Yaskawa INFORM job: R2_W02,4,6(0_0)_MP_OK.JBI

/JOB
//NAME R2_W02,4,6(0_0)_MP_OK
///FOLDERNAME MP_TEST
//POS
///NPOS 87,87,0,4,0,0
///TOOL 0
///POSTYPE PULSE
///PULSE
C00000=174522,6583,732,81114,57384,11781
C00001=174517,6598,745,81115,57387,11780
C00002=174515,6604,750,81115,57388,11780
C00003=173653,9147,2977,81262,57995,11683
C00004=173711,9248,3067,81257,57952,11686
C00005=173653,9147,2977,81262,57995,11683
C00006=174515,6604,750,81115,57388,11780
C00007=174498,6652,791,75592,65380,14408
C00008=174498,6652,791,75592,65380,14408
C00009=174498,6652,791,75592,65380,14408
C00010=176658,117,-15048,82463,49173,12368
C00011=174531,6571,721,88243,49982,8451
C00012=174533,6604,911,88329,49975,8393
C00013=174531,6571,721,88243,49982,8451
C00014=174523,6586,734,88244,49988,8450
C00015=174526,6579,728,88244,49987,8450
C00016=174531,6564,715,88243,49983,8451
C00017=160984,-11348,3930,36053,37207,-42708
C00018=160980,-11334,3941,36055,37209,-42709
C00019=160979,-11329,3945,36056,37210,-42710
C00020=161194,-11069,4145,35902,37129,-42610
C00021=160979,-11329,3945,36056,37210,-42710
C00022=160995,-11368,3914,36742,28122,-41255
C00023=160996,-11216,4319,36932,27985,-41352
C00024=160995,-11368,3914,36742,28122,-41255
C00025=160973,-11311,3958,34758,46261,-43992
C00026=160980,-11331,3943,34756,46258,-43990
C00027=160980,-11331,3943,34756,46258,-43990
C00028=160980,-11331,3943,34756,46258,-43990
C00029=160973,-11311,3958,34758,46261,-43992
C00030=160973,-11311,3958,34758,46261,-43992
C00031=160974,-11316,3955,34758,46261,-43992
C00032=160977,-11328,3945,34757,46259,-43991
C00033=155155,-6207,-30499,23040,84085,-41474
C00034=187974,16007,-465,74860,68606,73739
C00035=187971,16014,-459,74861,68608,73738
C00036=187970,16017,-457,74861,68609,73738
C00037=188065,16322,-175,74847,68538,73741
C00038=187970,16017,-457,74861,68609,73738
C00039=187982,15993,-478,74858,68601,73740
C00040=188123,15688,-759,74825,68507,73762
C00041=187982,15993,-478,74858,68601,73740
C00042=187982,15995,-476,74858,68601,73740
C00043=188055,16230,-74,74890,68512,73687
C00044=187982,15995,-476,74858,68601,73740
C00045=187983,15992,-479,74858,68601,73740
C00046=187985,15986,-485,74857,68599,73740
C00047=155155,-6207,-30499,23040,84085,-41474
C00048=161010,6792,897,39431,61770,-2600
C00049=161008,6803,906,39432,61771,-2600
C00050=161106,6439,785,39434,61637,-2607
C00051=161075,4879,-316,39487,61556,-2657
C00052=160508,6816,-113,39396,62494,-2543
C00053=161011,6899,1448,34591,61140,-1667
C00054=173294,-15772,-2365,19599,41502,-27150
C00055=174899,-11478,4010,19118,39501,-26768
C00056=174262,-12641,3696,19743,39267,-27176
C00057=174084,-11684,2460,19373,40493,-26971
C00058=174842,-11820,3581,23453,38073,-33209
C00059=174431,-11387,3914,23749,38204,-33407
C00060=174436,-11399,3906,23747,38202,-33405
C00061=174416,-11363,3933,23761,38209,-33414
C00062=155155,-6207,-30499,23040,84085,-41474
C00063=174170,40084,30970,44829,89709,-71753
C00064=174201,39824,30698,44830,89717,-71735
C00065=174202,39772,30629,44830,89729,-71730
C00066=174202,39771,30687,44829,89703,-71742
C00067=173753,38726,28593,44851,90472,-71609
C00068=173790,41778,32604,44829,89804,-71890
C00069=174284,39520,30698,43457,86472,-69264
C00070=174527,39515,30359,43444,86501,-69136
C00071=174215,39612,30410,43455,86673,-69209
C00072=174214,39663,30476,43455,86662,-69214
C00073=174184,39924,30747,43457,86653,-69232
C00074=155155,-6207,-30499,23040,84085,-41474
C00075=160633,-10270,5638,28338,22900,-47145
C00076=162219,-15798,1425,26285,22163,-46063
C00077=160659,-10505,5478,28325,22871,-47138
C00078=160661,-10727,4919,28067,23075,-47011
C00079=161098,-12444,3311,27327,23025,-46629
C00080=159658,-10599,5699,29947,23053,-47982
C00081=160917,-11163,4021,24405,19147,-46607
C00082=160969,-11372,4753,24990,18622,-46880
C00083=160661,-10807,5180,25528,18740,-47150
C00084=160656,-10808,5155,25519,18754,-47146
C00085=135615,-20366,-13260,37178,48093,-50762
C00086=15978,-102434,-83816,28834,48298,-44128
BC00000=388510,12234,707895
BC00001=380989,10464,701589
BC00002=377980,9756,699066
BC00003=377846,15,698926
BC00004=375507,15,698920
BC00005=377846,15,698926
BC00006=377980,9756,699066
BC00007=360773,4968,724258
BC00008=360752,2897,724236
BC00009=360773,4968,724258
BC00010=374300,26988,580273
BC00011=374300,26988,580273
BC00012=374302,26995,572208
BC00013=374300,26988,580273
BC00014=379137,9576,654055
BC00015=382103,10646,655203
BC00016=389520,13320,658072
BC00017=313352,46812,968569
BC00018=306234,44848,958660
BC00019=303387,44062,954697
BC00020=300998,44084,954691
BC00021=303387,44062,954697
BC00022=302385,72266,846935
BC00023=302386,72273,838870
BC00024=302385,72266,846935
BC00025=301794,28524,989445
BC00026=305297,28517,959783
BC00027=305280,26764,959765
BC00028=305297,28517,959783
BC00029=301794,28524,989445
BC00030=301708,28983,989449
BC00031=304507,29324,994442
BC00032=311505,30175,1006925
BC00033=296594,86442,873629
BC00034=388565,51804,658383
BC00035=383620,57007,647781
BC00036=381641,59088,643541
BC00037=379252,59110,643535
BC00038=381641,59088,643541
BC00039=390370,60897,618560
BC00040=390394,63201,618584
BC00041=390370,60897,618560
BC00042=388386,59719,612189
BC00043=388387,59726,604124
BC00044=388386,59719,612189
BC00045=390364,57638,616429
BC00046=395310,52435,627031
BC00047=296594,86442,873629
BC00048=313394,73469,855255
BC00049=307271,69988,843128
BC00050=304895,68636,838421
BC00051=304822,68595,838277
BC00052=304822,68595,838277
BC00053=308544,65120,825419
BC00054=314454,36752,936853
BC00055=314454,36752,936853
BC00056=314454,36752,936853
BC00057=314454,36752,936853
BC00058=323351,25201,911905
BC00059=326138,25881,916533
BC00060=333107,27583,928104
BC00061=333060,27580,1035638
BC00062=296594,86442,873629
BC00063=333324,97353,980736
BC00064=333273,97166,873204
BC00065=330544,102864,857707
BC00066=329453,105143,851509
BC00067=329453,105143,851509
BC00068=329453,105143,851509
BC00069=333744,110491,853540
BC00070=351310,110324,799899
BC00071=352593,108156,806169
BC00072=355802,102738,821843
BC00073=355852,102924,929375
BC00074=296594,86442,873629
BC00075=301704,63726,1065666
BC00076=301654,63540,958133
BC00077=294938,60391,948793
BC00078=292251,59131,945057
BC00079=292251,59131,945057
BC00080=292251,59131,945057
BC00081=289814,66040,921083
BC00082=289884,78172,833466
BC00083=292523,79582,836925
BC00084=299118,83106,845574
BC00085=299169,83292,953107
BC00086=277147,104204,968203
///POSTYPE BASE
///RECTAN
///RCONF 0,0,0,0,0,0,0,0,0,0,0,0,0,0,0,0,0,0,0,0,0,0,0,0
P00006=0.222,-3.123,-1.508,0.0000,0.0000,0.0000
P00021=-0.225,-6.128,-0.405,0.0000,0.0000,0.0000
P00024=0.145,-0.552,1.326,0.0000,0.0000,0.0000
P00026=0.562,-0.002,-0.337,0.0000,0.0000,0.0000
//INST
///DATE 2023/11/16 16:40
///ATTR SC,RW
///GROUP1 RB1,BS1
NOP
'r2_W02,4,6
'Path S702 (for W1)
SFTOF
MOVL C00000 BC00000 V=100.0
MOVL C00001 BC00001 V=100.0
MOVL C00002 BC00002 V=100.0
MOVL C00003 BC00003 V=60.0
REFP 3 C00004 BC00004
CALL JOB:SEARCH-R1
SET P021 P006
SFTON P021
MOVL C00005 BC00005 V=60.0
MOVL C00006 BC00006 V=100.0
MOVL C00007 BC00007 V=60.0
REFP 3 C00008 BC00008
CALL JOB:SEARCH-R1
SET P021 P006
SFTON P021
MOVL C00009 BC00009 V=60.0
MOVL C00010 BC00010 V=100.0
MOVL C00011 BC00011 V=60.0
REFP 3 C00012 BC00012
CALL JOB:SEARCH-R1
SET P021 P006
SFTON P021
MOVL C00013 BC00013 V=60.0
MOVL C00014 BC00014 V=100.0
MOVL C00015 BC00015 V=100.0
MOVL C00016 BC00016 V=100.0
'Path S708 (for W4)
SFTOF
MOVL C00017 BC00017 V=100.0
MOVL C00018 BC00018 V=100.0
MOVL C00019 BC00019 V=60.0
REFP 3 C00020 BC00020
CALL JOB:SEARCH-R1
SET P026 P006
SFTON P026
MOVL C00021 BC00021 V=60.0
MOVL C00022 BC00022 V=60.0
REFP 3 C00023 BC00023
CALL JOB:SEARCH-R1
SET P026 P006
SFTON P026
MOVL C00024 BC00024 V=60.0
MOVL C00025 BC00025 V=100.0
MOVL C00026 BC00026 V=60.0
REFP 3 C00027 BC00027
CALL JOB:SEARCH-R1
SET P026 P006
SFTON P026
MOVL C00028 BC00028 V=60.0
MOVL C00029 BC00029 V=100.0
MOVL C00030 BC00030 V=100.0
MOVL C00031 BC00031 V=100.0
MOVL C00032 BC00032 V=100.0
MOVJ C00033 BC00033 VJ=20.00
'Path S705 (for W3)
SFTOF
MOVL C00034 BC00034 V=100.0
MOVL C00035 BC00035 V=100.0
MOVL C00036 BC00036 V=60.0
REFP 3 C00037 BC00037
CALL JOB:SEARCH-R1
SET P024 P006
SFTON P024
MOVL C00038 BC00038 V=60.0
MOVL C00039 BC00039 V=60.0
REFP 3 C00040 BC00040
CALL JOB:SEARCH-R1
SET P024 P006
SFTON P024
MOVL C00041 BC00041 V=60.0
MOVL C00042 BC00042 V=60.0
REFP 3 C00043 BC00043
CALL JOB:SEARCH-R1
SET P024 P006
SFTON P024
MOVL C00044 BC00044 V=60.0
MOVL C00045 BC00045 V=100.0
MOVL C00046 BC00046 V=100.0
MOVJ C00047 BC00047 VJ=20.00
'Path W1
SFTOF
SFTON P021
MOVL C00048 BC00048 V=100.0
MOVL C00049 BC00049 V=100.0
MOVL C00050 BC00050 V=100.0 PL=0
REFP 1 C00051 BC00051
REFP 2 C00052 BC00052
MACRO1 MJ#(0) ARGF10
ARCON
MOVL C00053 BC00053 V=13.3
ARCOF
SFTOF
'Path W2
SFTOF
SFTON P021
MOVL C00054 BC00054 V=100.0
MOVL C00055 BC00055 V=100.0 PL=0
REFP 1 C00056 BC00056
REFP 2 C00057 BC00057
MACRO1 MJ#(0) ARGF10
ARCON
MOVL C00058 BC00058 V=13.3
ARCOF
MOVL C00059 BC00059 V=100.0
MOVL C00060 BC00060 V=100.0
MOVL C00061 BC00061 V=100.0
SFTOF
'
MOVJ C00062 BC00062 VJ=20.00
'Path W786
SFTOF
SFTON P024
MOVJ C00063 BC00063 VJ=20.00
MOVL C00064 BC00064 V=100.0
MOVL C00065 BC00065 V=100.0
MOVL C00066 BC00066 V=100.0 PL=0
REFP 1 C00067 BC00067
REFP 2 C00068 BC00068
MACRO1 MJ#(0) ARGF10
ARCON
MOVL C00069 BC00069 V=13.3
MOVL C00070 BC00070 V=13.3
ARCOF
MOVL C00071 BC00071 V=100.0
MOVL C00072 BC00072 V=100.0
MOVL C00073 BC00073 V=100.0
SFTOF
MOVJ C00074 BC00074 VJ=20.00
'
'Path W4
SFTOF
SFTON P026
MOVJ C00075 BC00075 VJ=20.00
MOVL C00076 BC00076 V=100.0
WAIT IG#(200)=21
MOVL C00077 BC00077 V=100.0
MOVL C00078 BC00078 V=100.0 PL=0
REFP 1 C00079 BC00079
REFP 2 C00080 BC00080
MACRO1 MJ#(0) ARGF10
ARCON
MOVL C00081 BC00081 V=13.3
MOVL C00082 BC00082 V=13.3
ARCOF
MOVL C00083 BC00083 V=100.0
MOVL C00084 BC00084 V=100.0
MOVL C00085 BC00085 V=100.0
MOVJ C00086 BC00086 VJ=20.00
SFTOF
END
